ABB RobotStudio station: CageTest.rsstnx

Station CageTest (saved by RobotStudio 25.1.11133.0)
Controller IRB1100
  mechanical unit ROB_1: IRB1100, 6 joints, base frame (0, 0, 0) mm
Layout (positions relative to the parent item):
  - 3 - OmniCore_C30 [part, from %ABB.RobotStudio.Models.OmniCore%\OmniCore_C30.rslib] at (670.2, -528.83, -372.02) mm, rotated rx 0 ry 0 rz 90 deg
  - 4 - OmniCore_FlexPendant [graphiccomponentgroup, from %ABB.RobotStudio.Models.OmniCore%\OmniCore_FlexPendant.rslib] at (785.94, -489.8, -90.59) mm, rotated rx 0 ry 0 rz 90 deg
    - FlexPendant [part, from %ABB.RobotStudio.Models.OmniCore%\OmniCore_FlexPendant.rslib] at (0, 0, 15.72) mm
    - Holder [part, from %ABB.RobotStudio.Models.OmniCore%\OmniCore_FlexPendant.rslib]
  - IRB1100 [mechanism, from %ABB.RobotStudio.Models.IRB1100%\IRB1100_4_58__02.rslib] at (0, 0, 0) mm; joint values [0.5013, 0.0773, 0, 0, 0.5236, 0] (rad or m)
  - 1 - EntireModelLamps--12-03-2025 [graphiccomponentgroup] at (688.73, -603.31, 117.65) mm, rotated rx 0 ry 0 rz 90 deg
    - node0 [part] at (0, -1.43, 0) mm, size 1310 x 1175 x 1885 mm
    - node1 [part], size 35 x 60 x 45 mm
    - node2 [part], size 35 x 60 x 45 mm
    - node3 [part], size 35 x 60 x 45 mm
    - node4 [part], size 30 x 50 x 45 mm
    - node5 [part], size 35 x 60 x 45 mm
    - node6 [part], size 35 x 60 x 45 mm
    - node7 [part], size 35 x 60 x 45 mm
    - node8 [part], size 35 x 60 x 45 mm
    - Highlighter_2 [smart component, from Components\Highlighter.rslib] at (603.31, 688.73, -117.65) mm, rotated rx 0 ry 0 rz -90 deg
        properties: Object=autoModeLamp; Color=[0 204 0]; Opacity=255
  - 2 - LampsDescriptionPlate [graphiccomponentgroup] at (691.23, 279.23, -59.91) mm, rotated rx 90 ry 0 rz 90 deg
    - node0 [part], size 490 x 45 x 8 mm
    - node1 [part], size 490 x 45 x 5 mm
  - programmableLamp [part] at (688.64, 474.23, -139.8) mm, rotated rx 0 ry 90 rz 0 deg, size 28 x 28 x 5 mm
  - autoModeLamp [part] at (689.1, 439.16, -140.01) mm, rotated rx 0 ry 90 rz 0 deg, size 28 x 28 x 5 mm
  - continousModeLamp [part] at (689.17, 404.15, -139.91) mm, rotated rx 0 ry 90 rz 0 deg, size 28 x 28 x 5 mm
  - startingOverLamp [part] at (688.61, 339.1, -140.06) mm, rotated rx 0 ry 90 rz 0 deg, size 28 x 28 x 5 mm
  - runningProgramLamp [part] at (688.92, 304.07, -139.94) mm, rotated rx 0 ry 90 rz 0 deg, size 28 x 28 x 5 mm
  - errorLamp [part] at (689.5, 269.14, -139.8) mm, rotated rx 0 ry 90 rz 0 deg, size 28 x 28 x 5 mm
  - motorsOnLamp [part] at (689.42, 234.14, -140.11) mm, rotated rx 0 ry 90 rz 0 deg, size 28 x 28 x 5 mm
  - 5 - lampsControl [smart component]
      signals: DI DI_AutoMode, DI DI_Error, DI DI_MotorsOn, DI DI_Program, DI DI_StartOver, DI DI_Continous, DI DI_ProgrammableLamp
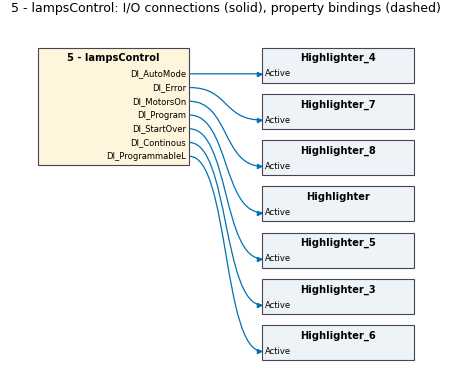
      connections:
        5 - lampsControl.DI_AutoMode -> Highlighter_4.Active
        5 - lampsControl.DI_Error -> Highlighter_7.Active
        5 - lampsControl.DI_MotorsOn -> Highlighter_8.Active
        5 - lampsControl.DI_Program -> Highlighter.Active
        5 - lampsControl.DI_StartOver -> Highlighter_5.Active
        5 - lampsControl.DI_Continous -> Highlighter_3.Active
        5 - lampsControl.DI_ProgrammableLamp -> Highlighter_6.Active
    - Highlighter [smart component, from Components\Highlighter.rslib]
        properties: Object=programmableLamp; Color=[255 255 255]; Opacity=255
    - Highlighter_3 [smart component, from Components\Highlighter.rslib]
        properties: Object=continousModeLamp; Color=[255 255 255]; Opacity=255
    - Highlighter_4 [smart component, from Components\Highlighter.rslib]
        properties: Object=autoModeLamp; Color=[0 204 0]; Opacity=255
    - Highlighter_5 [smart component, from Components\Highlighter.rslib]
        properties: Object=startingOverLamp; Color=[255 255 255]; Opacity=255
    - Highlighter_6 [smart component, from Components\Highlighter.rslib]
        properties: Object=runningProgramLamp; Color=[0 204 0]; Opacity=255
    - Highlighter_7 [smart component, from Components\Highlighter.rslib]
        properties: Object=errorLamp; Color=[255 128 0]; Opacity=255
    - Highlighter_8 [smart component, from Components\Highlighter.rslib]
        properties: Object=motorsOnLamp; Color=[0 204 0]; Opacity=255
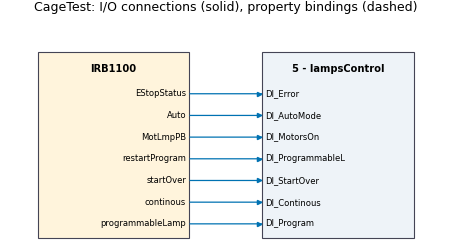
Station logic (signal -> signal, property => property):
  IRB1100.EStopStatus -> 5 - lampsControl.DI_Error
  IRB1100.Auto -> 5 - lampsControl.DI_AutoMode
  IRB1100.MotLmpPB -> 5 - lampsControl.DI_MotorsOn
  IRB1100.restartProgram -> 5 - lampsControl.DI_ProgrammableLamp
  IRB1100.startOver -> 5 - lampsControl.DI_StartOver
  IRB1100.continous -> 5 - lampsControl.DI_Continous
  IRB1100.programmableLamp -> 5 - lampsControl.DI_Program
Targets, tools, work objects and paths stored in the station, written as RAPID:
! task T_ROB1
MODULE Module1
  PROC main()
  ENDPROC
ENDMODULE

! task T_ROB1
MODULE Module1
  PROC main()
  ENDPROC
ENDMODULE

